// TIA Portal V17 export
// export: Created 2024-08-09T12:53:09.5881925Z, ExportSetting WithDefaults, DisplayName Totally Integrated Automation Portal, DisplayVersion V17 Update 7, DisplayName TIA Portal Openness, DisplayVersion V17 Update 7, DisplayName TIA Portal Version Control Interface, DisplayVersion V17, DisplayName STEP 7 Professional, DisplayVersion V17 Update 7, DisplayName STEP 7 Safety, DisplayVersion V17 Update 6, DisplayName WinCC Professional, DisplayVersion V17 Update 7
VAR_GLOBAL   // PLC tag table "Mobile"
END_VAR
VAR_GLOBAL CONSTANT   // user constants
   Nbr_Max_Mobiles : UInt := 499;   // Nombre maximal de mobiles
   Nbr_Max_Pos : USInt := 19;   // Nombre de positions possibles pour le mobile
   Nbr_Entr_Pos : USInt := 29;   // Nombre d'entrees a tester pour chaque position mobile
   Nbr_Sort_Pos : USInt := 9;   // Nombre de sorties a piloter pour chaque position mobile
   Nbr_Mob_Suiv : USInt := 19;   // Nombre de mobiles suivants possible
   Nbr_Mob_Prec : USInt := 19;   // Nombre de mobiles precedents possible
   Nbr_Mob_Horiz : USInt := 9;   // Nombre de mobiles horizontaux possible
   Ord_Pos : SInt := 0;   // Ordre de positionnement
   Ord_Fin_Pos : SInt := 1;   // Ordre de fin de positionnement
   Ord_Fin_Pos_Imm : SInt := 2;   // Ordre de fin positionnement immediatement
   Ord_Vid_Imm : SInt := 3;   // Ordre de vidange immediat
   HS : USInt := 0;   // Mobile hors service
   Libre : USInt := 1;   // Mobile libre: arrete
   Enc_Pos : USInt := 2;   // Mobile en cours de positionnement
   Pret : USInt := 3;   // Mobile pret
   Vid : USInt := 4;   // Mobile en vidange
   Mar_Force : USInt := 5;   // Mobile en marche forcee
   Enc_Fin_Pos : USInt := 6;   // Mobile en cours de fin positionnement
   Defaut : USInt := 7;   // Mobile en defaut
   Etp_Inactif : USInt := 0;   // Inactif
   Etp_Repos : USInt := 1;   // Attente demande de positionnement
   Etp_Test_Ent_Av_Pos : USInt := 2;   // Test des entrees avant positionnement
   Etp_Test_Verr : USInt := 3;   // Test disponibilite du mobile
   Etp_Att_Suiv_Pret : USInt := 4;   // Attente mobile suivant pret
   Etp_Positionnement : USInt := 5;   // Positionnement du mobile
   Etp_Surveillance : USInt := 6;   // Surveillance marche mobile
   Etp_Att_Fin_Pas_Mat : USInt := 7;   // Tempo maxi attente fin passage de la matiere
   Etp_Vidange : USInt := 8;   // Vidange du mobile
   Etp_Mar_For : USInt := 9;   // Marche forcee
   Etp_Fin_Pos_Imm : USInt := 10;   // Fin de positionnement immediat
   Etp_Test_Ent_Apr_Fin_Pos : USInt := 11;   // Test des entrees apres arret
   Etp_Tps_Apr_Fin_Pos : USInt := 12;   // Tempo imperative apres fin positionnement
   Etp_Tps_Av_Chang_Pos : USInt := 13;   // Tempo avant changement de position
   Etp_Chang_Pos : USInt := 14;   // Changement de position
   Etp_Chang_Mode : USInt := 15;   // Changement de mode
   Etp_Defaut : USInt := 16;   // Defaut mobile
   Etp_Att_Ack_Def : USInt := 17;   // Tempo imperative apres defaut
   Fct_Stock : USInt := 0;   // Fonction stockage silo
   Fct_Posit : USInt := 1;   // Fonction stockage Revolver
   PasDeCalcul : USInt := 16#0;   // Pas de calcul ni la qte ni leneregie[calc theo E,lire E direc , Calc ener oui non , calc qte oui nn]
   CalcQteSeul : USInt := 16#1;   // Calc de la quantite
   LireEnrjSeul : USInt := 16#6;   // Lire directement la valeur de l'energie
   CalcQteLireEnr : USInt := 16#7;   // Calc de la quantite et Lire directement la valeur de l'energie
   CalcEnrjSeul : USInt := 16#A;   // Calcul theor de l'energie
   CalcEnrjQte : USInt := 16#B;   // Calcul theor de l'energie et de la qte
END_VAR
